(* PLC project Tc3_EventLogger.SetJsonAttribute Demo, tc3-libraries-kb TwinCAT 3.1 *)
(* stored: creationDateTime 2026-05-11T01:00:00, modificationDateTime 2026-05-11T01:00:00 *)

PROGRAM P_Demo_FB_TcMessage_SetJsonAttribute
  VAR
    fbMessage : FB_TcMessage;  (* message 实例（已 Create） *)
    bSetAttr : BOOL := FALSE;  (* 上升沿触发 *)
    bSetAttrPrev : BOOL;  (* 边沿检测 *)
    sBatchId : STRING := 'B-2026-0511-001';  (* 批次号 *)
    sJsonAttribute : STRING;  (* 拼接好的完整 JSON *)
    hr : HRESULT;  (* 返回值监视 *)
  END_VAR

// =============================================================================
// 场景：配方切换消息附加批次追溯 JSON
// 价值：一句调用绑定上下文到 message
// 验证：登录后写 bSetAttr := TRUE，HMI 事件详情应能看到 JSON 字段
// 验证步骤：
//   1. 右键 PLC 项目 → Import PLCopenXML → 选本文件
//   2. 引用 Tc3_EventLogger（System → References → Add library）
//   3. 编译 → 登录 → 运行；按 verify 注释里给出的在线写值操作
// =============================================================================

sJsonAttribute := CONCAT('{"batch":"', CONCAT(sBatchId, '"}'));

IF bSetAttr AND NOT bSetAttrPrev THEN
    hr := fbMessage.SetJsonAttribute(sJsonAttribute := sJsonAttribute);
END_IF;
bSetAttrPrev := bSetAttr;
END_PROGRAM
